(* PLC project  *)

PROGRAM P
  VAR  (* added by the conversion: wires and edge detectors of the diagram *)
    _F_X3_R : ANY;
    _F_X3_OUT : ANY;
  END_VAR

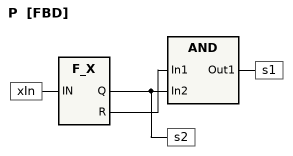
(* FBD diagram, written out as Structured Text *)
_F_X3_OUT := F_X(IN := xIn, R => _F_X3_R);
s2 := _F_X3_OUT;
s1 := _F_X3_R AND _F_X3_OUT;
END_PROGRAM
